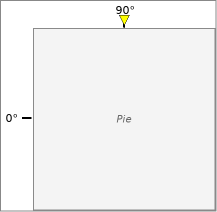
VISUALIZATION VISU_Tube_Side  // 217x212
VAR_IN_OUT
	ele : LREAL;
    eleTarget : LREAL;
    eleTargetInvisible : BOOL;
    mark10Degrees : LREAL;
END_VAR
    Polyline (124,31) (124,51)
        p2858320360: ele
    Polygon (101,153) (147,153) (147,42) (101,42)
        p2858320360: ele
    Ellipse (88,83 71x71)
    Ellipse (91,86 65x65)
    Polygon (130,114) (130,126) (157,119) (157,117)
    Polygon (118,114) (130,114) (125,85) (123,85)
    Polygon (118,114) (118,126) (90,119) (90,117)
    Polygon (85,176) (93,176) (105,128) (97,128)
    Polygon (154,176) (162,176) (150,128) (142,128)
    Polygon (93,176) (154,176) (142,128) (105,128)
    Ellipse (114,110 19x19)
    Polygon (119,37) (124,27) (129,37)
        p2858320360: ele
    Polygon (127,145) (138,145) (138,157) (127,157)
    Pie (33,28 182x182)
    Polyline (124,27) (124,18)
    Rectangle (110,3 31x15), "90°"
    Polyline (31,118) (22,118)
    Rectangle (2,111 20x15), "0°"
    Polyline (124,27) (124,22)
        p2858320360: -10
    Polyline (124,27) (124,22)
        p2858320360: -20
    Polyline (124,27) (124,22)
        p2858320360: -30
    Polyline (124,27) (124,22)
        p2858320360: -40
    Polyline (124,27) (124,22)
        p2858320360: -50
    Polyline (124,27) (124,22)
        p2858320360: -60
    Polyline (124,27) (124,22)
        p2858320360: -70
    Polyline (124,27) (124,22)
        p2858320360: -80
    Polygon (119,15) (124,25) (129,15), invisible if: eleTargetInvisible
        p2858320360: eleTarget
END_VISUALIZATION

(* stored: Version 1.1.0.1, ProductVersion 3.1.4019.2
   Visu VISU_Tube_Side: Id {5bb00c13-432c-4434-b0bb-547166592679} *)
